FUNCTION_BLOCK TemplateSimple (* Simple FB with one algorithm *)
  (* Standard: 61499-1 *)
  (* Version 0.0, 2018-10-15, Peter Gsellmann, TU Wien/ACIN *)
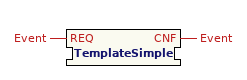
  EVENT_INPUT
    REQ; (* Normal Execution Request *)
  END_EVENT
  EVENT_OUTPUT
    CNF; (* Execution Confirmation *)
  END_EVENT
  EC_STATES
    REQ : REQ -> CNF;
  END_STATES
  ALGORITHM REQ IN ST:

  END_ALGORITHM
END_FUNCTION_BLOCK
